// TIA Portal V18 export
DATA_BLOCK "deleteeeaman_sel_target_DB"   // DB52
VERSION : 0.1
// stored: AutoNumber true, DBAccessibleFromOPCUA true, InstanceOfName aman_sel_target, InstanceOfType FB
"aman_sel_target"
   // VAR_INPUT
   //    allowed : Bool;
   //    team_unison : Bool;
   //    team_free : Bool;
   //    team_override : Bool;
   //    xbtnAnyMan : Bool;
   //    xbtnHome : Bool;
   //    xbtnStepPlus : Bool;
   //    xbtnStepMinus : Bool;
   //    execUni : Bool;
   //    targetUni : Real;
   //    targetHome : Real;
   //    targetStep : Real;
   //    POS : Real;
   // END_VAR
   // VAR_OUTPUT
   //    ExecuteSemiAutoManuver : Bool;
   //    m_auto : Bool;
   //    m_man : Bool;
   //    m_override : Bool;
   //    target : Real;
   //    execute : Bool;
   // END_VAR
   // VAR
   //    auto_allowed : Bool;
   //    anyBtn : Bool;
   //    xbtnHome_was : Bool;
   //    bsuhome { S7_SetPoint := 'True'} : "_ML2_ts_block1_subunit";
   //    p1Home : Bool;
   //    q1Home : Bool;
   //    Q_integer : Int;
   //    bsu_step_plus { S7_SetPoint := 'True'} : "_ML2_ts_block1_subunit";
   //    p2StepPlus : Bool;
   //    q2StepPlus : Bool;
   //    p3StepMinus : Bool;
   //    q3StepMinus : Bool;
   //    bsu_step_minus { S7_SetPoint := 'True'} : "_ML2_ts_block1_subunit";
   // END_VAR
BEGIN
END_DATA_BLOCK
